FUNCTION_BLOCK 22
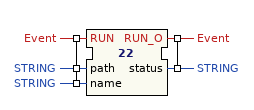
  EVENT_INPUT
    RUN WITH path, name;
  END_EVENT
  EVENT_OUTPUT
    RUN_O WITH status;
  END_EVENT
  VAR_INPUT
    path : STRING;
    name : STRING;
  END_VAR
  VAR_OUTPUT
    status : STRING;
  END_VAR
END_FUNCTION_BLOCK
